Staubli VAL3: Entwicklungsmethodik.dtx

mdesc mNomSpeed
frame fUserFrame = {x=701.757897, y=-321.609007, z=-207.673108, rx=-0.0947033, ry=0.52905, rz=90.111007, fatherId=world[0]}
tool tGreifer = {x=1.13686837721616E-13, y=-4.40536496171262E-13, z=110.500000000003, rx=-1.59027734073174E-14, ry=3.10104081442691E-14, rz=-2.14687465591809E-14, fatherId=flange[0], ioLink=ValveIO\valve1, ioOpen=0.05, ioClose=0.05}
pointRx pABPosition[12]
  [0] = {x=100, y=100, z=20, rx=180, rz=45, fatherId=fUserFrame[0]}
  [1] = {x=200, y=100, z=20, rx=180, rz=45, fatherId=fUserFrame[0]}
  [2] = {x=300, y=100, z=20, rx=180, rz=45, fatherId=fUserFrame[0]}
  [3] = {x=400, y=100, z=20, rx=180, rz=45, fatherId=fUserFrame[0]}
  [4] = {x=100, y=200, z=20, rx=180, rz=45, fatherId=fUserFrame[0]}
  [5] = {x=200, y=200, z=20, rx=180, rz=45, fatherId=fUserFrame[0]}
  [6] = {x=300, y=200, z=20, rx=180, rz=45, fatherId=fUserFrame[0]}
  [7] = {x=400, y=200, z=20, rx=180, rz=45, fatherId=fUserFrame[0]}
  [8] = {x=100, y=300, z=20, rx=180, rz=45, fatherId=fUserFrame[0]}
  [9] = {x=200, y=300, z=20, rx=180, rz=45, fatherId=fUserFrame[0]}
  [10] = {x=300, y=300, z=20, rx=180, rz=45, fatherId=fUserFrame[0]}
  [11] = {x=400, y=300, z=20, rx=180, rz=45, fatherId=fUserFrame[0]}
sio soTcpClient = {link=Socket\server0}
bool bNewData[2]
num nData[3]
bool bReady
jointRx jHome = {j3=90, j5=90}
mdesc mUsedSpeed
pointRx pPick = {z=20, rx=180, rz=45, fatherId=fUserFrame[0]}
trsf trApro = {z=-150}
pointRx pPlace = {z=20, rx=180, rz=45, fatherId=fUserFrame[0]}
bool bPick
num nX
num nY
